{attribute 'qualified_only'}
VAR_GLOBAL
	fWinchValveOut : LREAL;
	fCylValveOut : LREAL;
END_VAR

(* stored: Version 1.1.0.1, ProductVersion 3.1.4024.12
   GVL NormalizedOutputs: Id {f796c89b-1bae-4f99-ace1-52ec7a3f08d2} *)
